// SIMATIC S7-200 project (STEP 7-Micro/WIN), CPU 224XP REL 02.01

SYMBOL_TABLE USER1
star             I0.0
stops            I0.1
den_1            Q0.0
den_2            Q0.1
den_3            Q0.2
den_4            Q0.3
den_5            Q0.4
bien_trung_gian  M0.0
den_6            Q0.5
den_7            Q0.6
den_8            Q0.7
den_9            Q1.0
den_10           Q1.1
END_SYMBOL_TABLE

ORGANIZATION_BLOCK MAIN:OB1
TITLE=PROGRAM COMMENTS
BEGIN
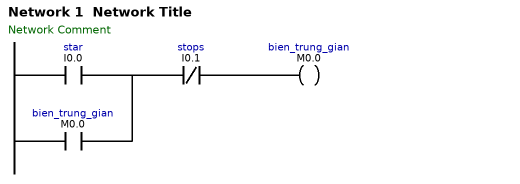
Network 1 // Network Title
// Network Comment
LD     star:I0.0
O      bien_trung_gian:M0.0
AN     stops:I0.1
=      bien_trung_gian:M0.0
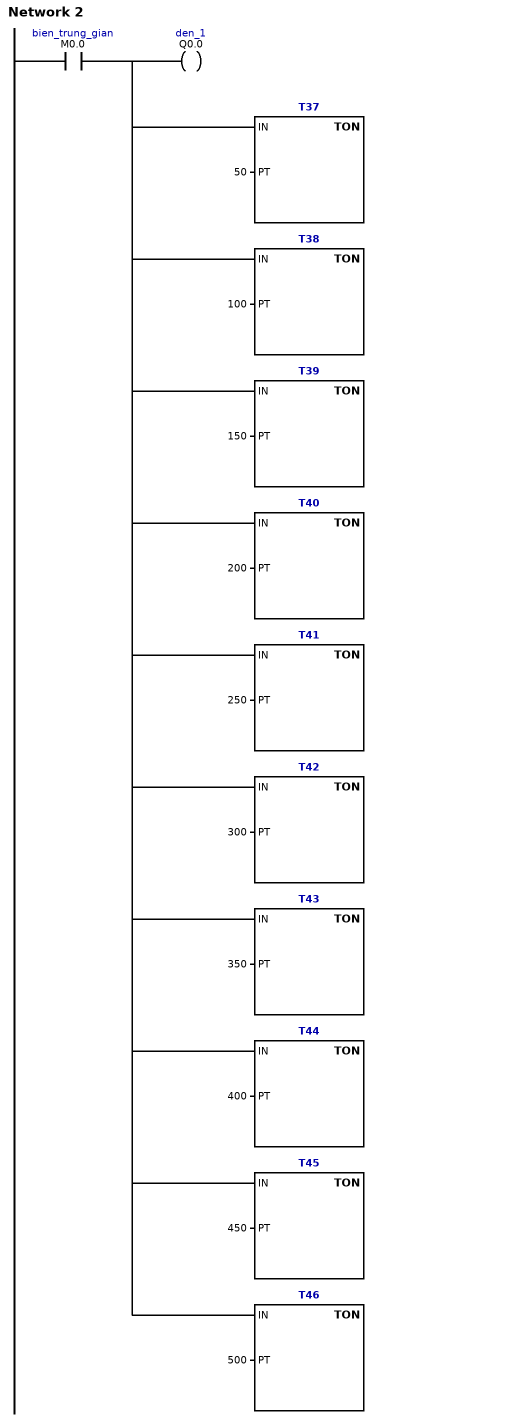
Network 2
LD     bien_trung_gian:M0.0
=      den_1:Q0.0
TON    T37, 50
TON    T38, 100
TON    T39, 150
TON    T40, 200
TON    T41, 250
TON    T42, 300
TON    T43, 350
TON    T44, 400
TON    T45, 450
TON    T46, 500
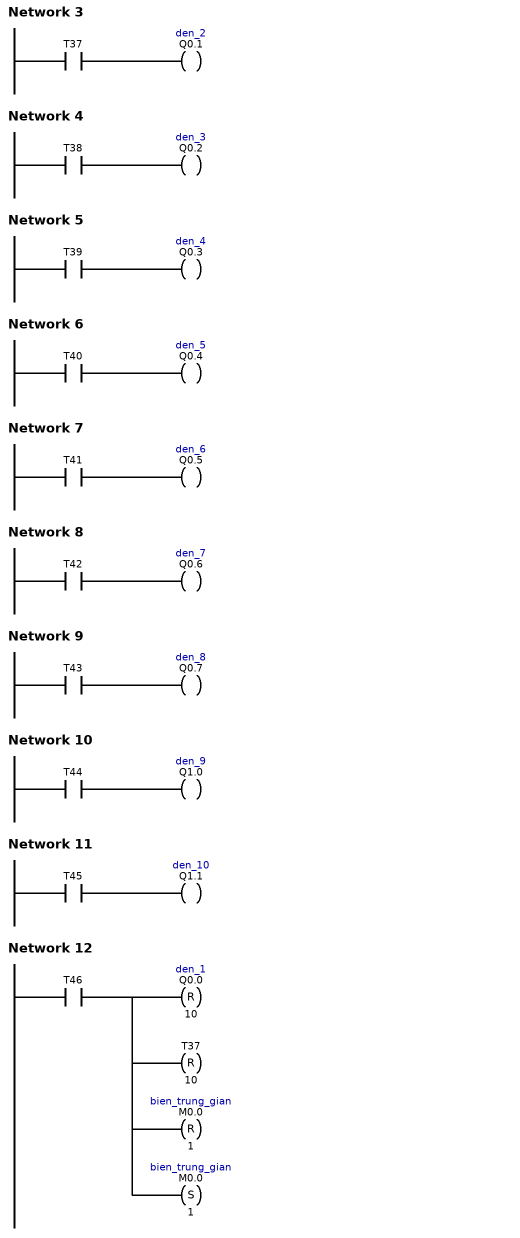
Network 3
LD     T37
=      den_2:Q0.1
Network 4
LD     T38
=      den_3:Q0.2
Network 5
LD     T39
=      den_4:Q0.3
Network 6
LD     T40
=      den_5:Q0.4
Network 7
LD     T41
=      den_6:Q0.5
Network 8
LD     T42
=      den_7:Q0.6
Network 9
LD     T43
=      den_8:Q0.7
Network 10
LD     T44
=      den_9:Q1.0
Network 11
LD     T45
=      den_10:Q1.1
Network 12
LD     T46
R      den_1:Q0.0, 10
R      T37, 10
R      bien_trung_gian:M0.0, 1
S      bien_trung_gian:M0.0, 1
END_ORGANIZATION_BLOCK
